FUNCTION_BLOCK LinearContinuousDrive_2Sensor EXTENDS FBA_LinearDrive IMPLEMENTS I_LinearContinuousDrive
VAR_INPUT
	drive : I_ContinuousDrive;
END_VAR
VAR
	extendLimit AT %I* : BOOL;
END_VAR

override();

ready := bEnable AND NOT Active AND HomeSet;

PROPERTY Active : BOOL
GET
Active := drive.Active;
END_GET
END_PROPERTY

PROPERTY AtExtendLimit : BOOL
GET
AtExtendLimit := extendLimit <> sensorDefaultState;
END_GET
END_PROPERTY

PROPERTY Error : BOOL
GET
error := drive.Error;
END_GET
END_PROPERTY

METHOD homingSequence : BOOL
(*
homing sequence is different for linear motion devices with limit sensors
*)
CASE step OF
	Homing.IDLE:
		reset();
		IF bEnable THEN
			step := Homing.START;
		END_IF
		
	Homing.START:
		IF AtHome THEN
			step := Homing.STOP;
			
		ELSIF AtExtendLimit THEN
			step := Homing.RETRY;
			
		ELSE
			moveContinuous(newDirection:= MC_Positive_Direction);
		END_IF
		
	Homing.STOP:
		IF stop() THEN
			step := Homing.DONE;
		END_IF
		
	Homing.DONE:
		homingComplete := TRUE;
		step := Homing.IDLE;
		
END_CASE
END_METHOD

METHOD moveContinuous : BOOL
VAR_INPUT
	newDirection : MC_Direction;
END_VAR
drive.moveContinuous(newDirection:= newDirection);

direction := newDirection;
END_METHOD

METHOD PRIVATE override : BOOL
VAR_INPUT
END_VAR
(*
-at home and attempting to traverse outward
-at outer limit and attempting to traverse outward
-at inner limit and attempting to traverse inwards
*)
(*
inward = negative direction, negative velocity
outward = positive direction, positive velocity
*)

IF error THEN
	stop();
	reset();
	
ELSIF
	(AtExtendLimit AND direction = MC_Negative_Direction) OR
	(AtHome AND direction = MC_Positive_Direction)
THEN
	stop();
END_IF
END_METHOD

METHOD reset : BOOL
VAR_INPUT
END_VAR
reset := drive.reset();
END_METHOD

METHOD stop : BOOL
VAR_INPUT
END_VAR
stop := drive.stop();
END_METHOD

METHOD toHome : BOOL
VAR_INPUT
END_VAR
IF AtHome THEN
	toHome := TRUE;
ELSE
	moveContinuous(newDirection := MC_Negative_Direction);
END_IF
END_METHOD

END_FUNCTION_BLOCK

(* stored: Version 1.1.0.1, ProductVersion 3.1.4024.11
   POU LinearContinuousDrive_2Sensor: Id {69fe43b2-faf3-4bb9-a151-1d9c1d256498}, SpecialFunc None
   Folder Private: Id {9b830d23-e10f-4ade-b1c6-bd40d8680072}
   Folder Properties: Id {222c607c-1a87-41f2-a4e5-82d9575d5282}
   Property Active: Id {be3c8ec3-3c7f-4ef3-ac2b-012ebbb0b2f4}
   Get Get: Id {bce40158-8ba9-497b-a2a4-eaedb5ee94af}
   Property AtExtendLimit: Id {9556aa23-042e-4218-90ac-c927b0a199c6}
   Get Get: Id {6a526c99-1448-4b8b-a742-5ed1740b7567}
   Property Error: Id {9da55b98-7c92-49b9-b94b-403edbd91f21}
   Get Get: Id {a1cb840b-6a4a-4350-9be9-67184bf97d67}
   Method homingSequence: Id {b1172124-9cb3-497c-8ea6-edcec54788c3}
   Method moveContinuous: Id {d3d7b24b-9b3b-4f48-8637-900b925c5f61}
   Method override: Id {10aaa485-7a7e-4baf-81f4-bb828e6d87bb}
   Method reset: Id {526a6cac-c4ab-4df7-9238-02b6edf9c7b5}
   Method stop: Id {82349e59-39b6-4b02-aab4-9afca6aa6f2f}
   Method toHome: Id {89aaf450-da88-4a41-a973-69fc801eb5bf} *)
